PROGRAM MAIN
VAR
	wEcMasterDevID AT %I*		:WORD;
	fbGetData_Coupler	 		:FB_GetMyLocalData;
	stSlaveInfo_Coupler 		:ST_SlaveInfo;
END_VAR

(* Example main program to show how to incorporate the VLS motion program *)

(*in stSlaveInfo is all information for getting current topology data
even if they changed by HotConnect*)
fbGetData_Coupler(wEcMasterDevID:= wEcMasterDevID, stSlaveInfo=>stSlaveInfo_Coupler );

IF stSlaveInfo_Coupler.bDataOk THEN // we are connected
	PRG_VLS_MOTION(); // So, run the program associated with coupler
END_IF

END_PROGRAM

(* stored: Version 1.1.0.1, ProductVersion 3.1.4024.2
   POU MAIN: Id {e6fa2b58-86f6-4521-8196-c6010dfb509b}, SpecialFunc None *)
